// TIA Portal V17 export
// export: Created 2025-03-07T09:24:11.3125459Z, ExportSetting WithDefaults, DisplayName Totally Integrated Automation Portal, DisplayVersion V17 Update 8, DisplayName TIA Portal Openness, DisplayVersion V17 Update 8, DisplayName TIA Portal Version Control Interface, DisplayVersion V17, DisplayName SINAMICS Startdrive Advanced, DisplayVersion V17 SP2, DisplayName SINAMICS Startdrive G110M, G120, G120C, G120D, G120P, G115D, DisplayVersion V17 SP2, DisplayName SINAMICS Startdrive G130, G150, S120, S150, SINAMICS MV, S210, DisplayVersion V17 SP2, DisplayName STEP 7 Professional, DisplayVersion V17 Update 8, DisplayName SINUMERIK ONE STEP 7 Toolbox, DisplayVersion V17 Update 12, DisplayName SINUMERIK 840D sl STEP 7 Toolbox, DisplayVersion V17 Update 12, DisplayName STEP 7 Safety, DisplayVersion V17 Update 6, DisplayName WinCC Advanced, DisplayVersion V17 Update 8
DATA_BLOCK "DB22108_HOPPER_LOWER_PART_TEMP_HOPPER_1_UNIT_01"   // DB22108
{ DB_Accessible_From_OPC_UA := 'FALSE' }
VERSION : 0.1
// stored: AutoNumber false, DBAccessibleFromOPCUA false, DBAccessibleFromWebserver true, InstanceOfName FB22104_TEMPERATURE_SENSOR, InstanceOfType FB
"FB22104_TEMPERATURE_SENSOR"
   // VAR_INPUT
   //    iANALOG_INPUT : Int;
   //    iCLEAR_LOG : Bool;
   // END_VAR
   // VAR_OUTPUT
   //    oERROR_LIMIT : Bool;
   //    oWARNING_LIMIT : Bool;
   // END_VAR
   // VAR
   //    OUTPUT : Struct
   //       VALUE : Real;
   //    END_STRUCT;
   //    INPUT_SETTINGS : Struct
   //       MAX_INPUT_VALUE : Real;
   //       IS_ANALOG_VALUE : Bool;
   //       UNIT_NUMBER : Int := 1;
   //       HOPPER_NUMBER : Int := 1;
   //    END_STRUCT;
   //    ALARMS_SETTINGS : Struct
   //       WARN_LIM_HIGH : Real;
   //       ERROR_LIM_HIGH : Real;
   //       WARN_LIM_LOW : Real;
   //       ERROR_LIM_LOW : Real;
   //       ERROR_CONFIGURATION : Bool;
   //    END_STRUCT;
   //    LOG : Struct
   //       MAX_TEMP_DATE : Date_And_Time;
   //       MAX_TEMP : Real;
   //    END_STRUCT;
   //    INTERNAL : Struct
   //       ERROR_CODE_T : Int;
   //       AUX : Bool;
   //    END_STRUCT;
   // END_VAR
BEGIN
END_DATA_BLOCK
